PROGRAM LLD
VAR
	i : INT := 0;
	f : REAL := 0.0;
	elapsed : TIME := TIME#0M0S0MS;
	today : DATE := DATE#2023-05-19;
	message : STRING := '';
	count : BYTE := 0;
	
	A AT %I* : BOOL := FALSE;
	B AT %I* : BOOL := FALSE;
	C AT %I* : BOOL := FALSE;
	D AT %Q* : BOOL := FALSE;
	
	op1 : INT := 1;
	op2 : INT := 2;
	res : REAL := 0.0;
	test : BOOL := FALSE;
	
	TON_0 : TON;
END_VAR

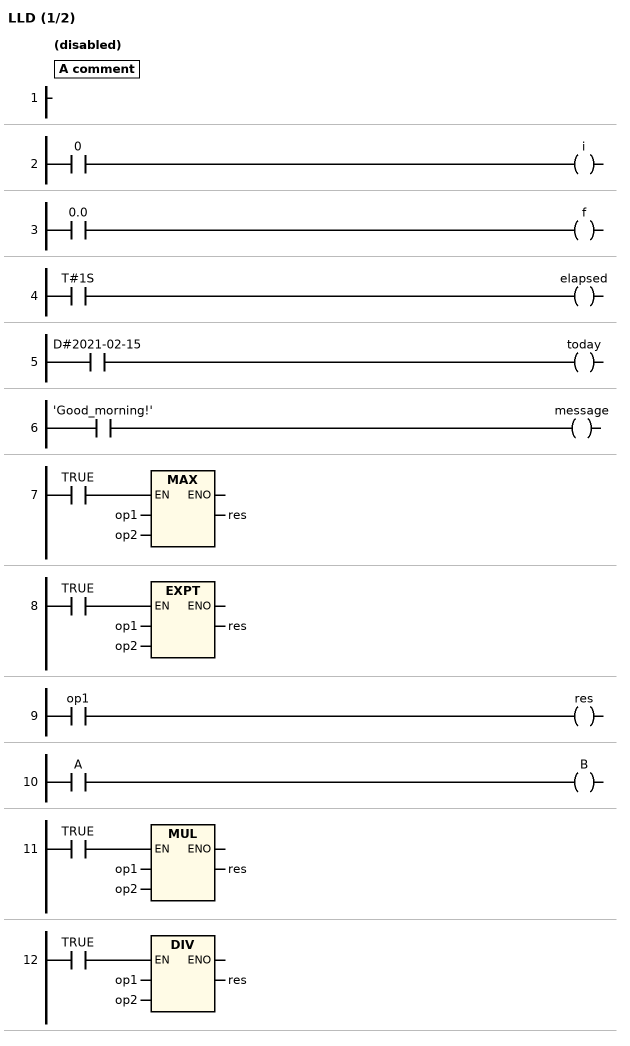
// NETWORK 1 (disabled)
// label: A comment

// NETWORK 2
i := 0;

// NETWORK 3
f := 0.0;

// NETWORK 4
elapsed := T#1S;

// NETWORK 5
today := D#2021-02-15;

// NETWORK 6
message := 'Good_morning!';

// NETWORK 7
res := MAX(op1, op2);

// NETWORK 8
res := EXPT(op1, op2);

// NETWORK 9
res := op1;

// NETWORK 10
B := A;

// NETWORK 11
res := op1 * op2;

// NETWORK 12
res := op1 / op2;

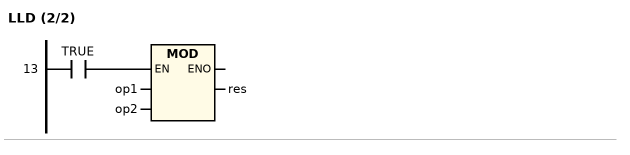
// NETWORK 13
res := op1 MOD op2;

END_PROGRAM

(* stored: Version 1.1.0.1, ProductVersion 3.1.4024.12
   POU LLD: Id {9db0e6b2-776d-446a-9237-26a0014307a9}, SpecialFunc None *)
